SUBAPPLICATION Uebung_028a (* Analog-Eingang *)
  (* Standard: 61499-2; Description: Copyright (c) 2023 Meisterschulen am Ostbahnhof This program and the accompanying materials are made available under the terms of the Eclipse Public License 2.0 which is available at https://www.eclipse.org/legal/epl-2.0/ SPDX-License-Identifier: EPL-2.0 *)
  (* Version 1.0, 2023-10-23, Franz Höpfinger, Meisterschulen am Ostbahnhof, initial API and implementation and/or initial documentation *)
  PACKAGE Uebungen;
  IMPORT logiBUS::io::DI::logiBUS_DI::Input_I1;
  IMPORT logiBUS::io::DI::logiBUS_DI::Input_I2;
  IMPORT logiBUS::io::DI::logiBUS_DI::Input_I3;
  IMPORT logiBUS::io::DI::logiBUS_DI_Events::BUTTON_SINGLE_CLICK;
  IMPORT logiBUS::io::DQ::logiBUS_DO::Output_Q1;
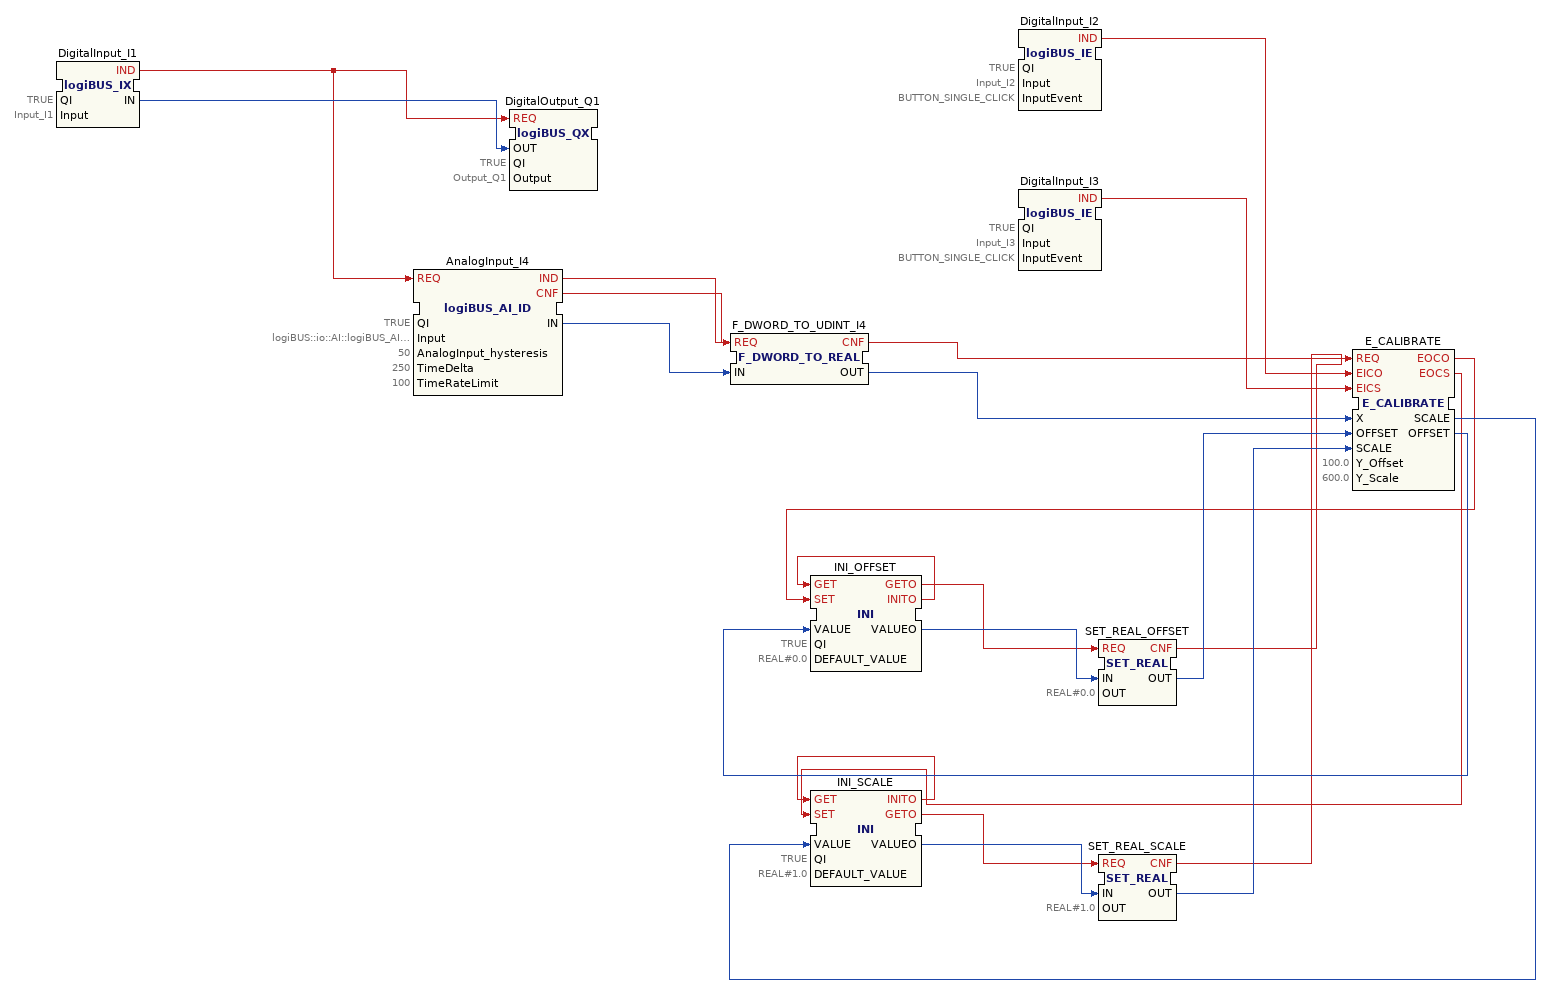
  FBS
    DigitalOutput_Q1 : logiBUS::io::DQ::logiBUS_QX(QI := TRUE, Output := Output_Q1);
    DigitalInput_I1 : logiBUS::io::DI::logiBUS_IX(QI := TRUE, Input := Input_I1);
    AnalogInput_I4 : logiBUS::io::AI::logiBUS_AI_ID(QI := TRUE, Input := logiBUS::io::AI::logiBUS_AI::AnalogInput_I4, AnalogInput_hysteresis := 50, TimeDelta := 250, TimeRateLimit := 100);
    F_DWORD_TO_UDINT_I4 : iec61131::conversion::F_DWORD_TO_REAL;
    E_CALIBRATE : OSCAT::Basic::POUs::Engineering::measurements::E_CALIBRATE(Y_Offset := 100.0, Y_Scale := 600.0);
    DigitalInput_I2 : logiBUS::io::DI::logiBUS_IE(QI := TRUE, Input := Input_I2, InputEvent := BUTTON_SINGLE_CLICK);
    DigitalInput_I3 : logiBUS::io::DI::logiBUS_IE(QI := TRUE, Input := Input_I3, InputEvent := BUTTON_SINGLE_CLICK);
    INI_OFFSET : eclipse4diac::storage::INI(QI := TRUE, DEFAULT_VALUE := REAL#0.0);
    SET_REAL_OFFSET : logiBUS::utils::conversion::provide::SET_REAL(OUT := REAL#0.0);
    INI_SCALE : eclipse4diac::storage::INI(QI := TRUE, DEFAULT_VALUE := REAL#1.0);
    SET_REAL_SCALE : logiBUS::utils::conversion::provide::SET_REAL(OUT := REAL#1.0);
  END_FBS
  EVENT_CONNECTIONS
    DigitalInput_I1.IND TO DigitalOutput_Q1.REQ;
    AnalogInput_I4.IND TO F_DWORD_TO_UDINT_I4.REQ;
    DigitalInput_I1.IND TO AnalogInput_I4.REQ;
    AnalogInput_I4.CNF TO F_DWORD_TO_UDINT_I4.REQ;
    F_DWORD_TO_UDINT_I4.CNF TO E_CALIBRATE.REQ;
    INI_OFFSET.GETO TO SET_REAL_OFFSET.REQ;
    INI_OFFSET.INITO TO INI_OFFSET.GET;
    INI_SCALE.INITO TO INI_SCALE.GET;
    INI_SCALE.GETO TO SET_REAL_SCALE.REQ;
    SET_REAL_OFFSET.CNF TO E_CALIBRATE.REQ;
    SET_REAL_SCALE.CNF TO E_CALIBRATE.REQ;
    DigitalInput_I2.IND TO E_CALIBRATE.EICO;
    DigitalInput_I3.IND TO E_CALIBRATE.EICS;
    E_CALIBRATE.EOCO TO INI_OFFSET.SET;
    E_CALIBRATE.EOCS TO INI_SCALE.SET;
  END_CONNECTIONS
  DATA_CONNECTIONS
    DigitalInput_I1.IN TO DigitalOutput_Q1.OUT;
    AnalogInput_I4.IN TO F_DWORD_TO_UDINT_I4.IN;
    F_DWORD_TO_UDINT_I4.OUT TO E_CALIBRATE.X;
    INI_OFFSET.VALUEO TO SET_REAL_OFFSET.IN;
    SET_REAL_OFFSET.OUT TO E_CALIBRATE.OFFSET;
    INI_SCALE.VALUEO TO SET_REAL_SCALE.IN;
    SET_REAL_SCALE.OUT TO E_CALIBRATE.SCALE;
    E_CALIBRATE.SCALE TO INI_SCALE.VALUE;
    E_CALIBRATE.OFFSET TO INI_OFFSET.VALUE;
  END_CONNECTIONS
END_SUBAPPLICATION
